// TIA Portal project "babu_3MotorsUsingComparatorsCounters" (V15)

(* hardware
DEVICE "S7-1200 station_1"  S7-1200 Station
   slot 0: "Rack_0"  S7-1200 Rack  Rack  V1.0
   slot 1: "PLC_1"  CPU 1212C DC/DC/DC  6ES7 212-1AE40-0XB0  V4.2
*)

// ===== PLC "PLC_1"  CPU 1212C DC/DC/DC =====

VAR_GLOBAL   // PLC tag table "Default tag table"
   "POWER ON PUSH BUTTON" AT %M0.0 : Bool;
   "POWER ON MEM" AT %M0.1 : Bool;
   "PULSE" AT %M0.2 : Bool;
   "RESTART PULSE" AT %M0.3 : Bool;
   "CYCLE COMPLETE" AT %M0.4 : Bool;
   "RESET COUNTER" AT %M0.5 : Bool;
END_VAR

// folder: System blocks/Program resources

DATA_BLOCK "IEC_Timer_0_DB"   // DB1
{ S7_Optimized_Access := 'TRUE' }
AUTHOR : Simatic
FAMILY : IEC
NAME : IEC_TMR
VERSION : 1.0
// stored: InstanceOfName IEC_TIMER
"IEC_TIMER"
BEGIN
END_DATA_BLOCK

DATA_BLOCK "IEC_Timer_0_DB_1"   // DB2
{ S7_Optimized_Access := 'TRUE' }
AUTHOR : Simatic
FAMILY : IEC
NAME : IEC_TMR
VERSION : 1.0
// stored: InstanceOfName IEC_TIMER
"IEC_TIMER"
BEGIN
END_DATA_BLOCK

DATA_BLOCK "IEC_Counter_0_DB"   // DB3
{ S7_Optimized_Access := 'TRUE' }
AUTHOR : Simatic
FAMILY : IEC
NAME : CNTR
VERSION : 1.0
// stored: InstanceOfName IEC_COUNTER
"IEC_COUNTER"
BEGIN
END_DATA_BLOCK

DATA_BLOCK "IEC_Timer_0_DB_2"   // DB4
{ S7_Optimized_Access := 'TRUE' }
AUTHOR : Simatic
FAMILY : IEC
NAME : IEC_TMR
VERSION : 1.0
// stored: InstanceOfName IEC_TIMER
"IEC_TIMER"
BEGIN
END_DATA_BLOCK

// folder: (top level)

ORGANIZATION_BLOCK "Main"   // OB1, LAD, ProgramCycle
TITLE = "Main Program Sweep (Cycle)"
{ S7_Optimized_Access := 'TRUE' }
VERSION : 0.1
   VAR_INPUT
      Initial_Call : Bool;   // Initial call of this OB
      Remanence : Bool;   // =True, if remanent data are available
   END_VAR
BEGIN

REGION Network 1
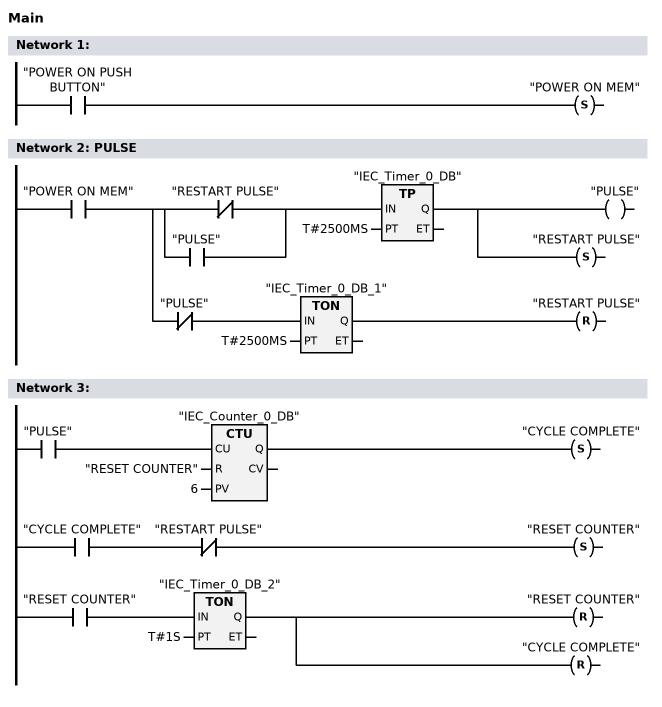
   RUNG wire#powerrail
      Contact( "POWER ON PUSH BUTTON" )
      S_Coil( "POWER ON MEM" )
   END_RUNG
   // the same network as SCL:
   IF "POWER ON PUSH BUTTON" THEN "POWER ON MEM" := TRUE; END_IF;
END_REGION

REGION Network 2: PULSE
   "IEC_Timer_0_DB".TP(IN := "POWER ON MEM" AND (NOT "RESTART PULSE" OR "PULSE"), PT := T#2500MS);
   "PULSE" := "IEC_Timer_0_DB".Q;
   IF "IEC_Timer_0_DB".Q THEN "RESTART PULSE" := TRUE; END_IF;
   "IEC_Timer_0_DB_1".TON(IN := "POWER ON MEM" AND NOT "PULSE", PT := T#2500MS);
   IF "IEC_Timer_0_DB_1".Q THEN "RESTART PULSE" := FALSE; END_IF;
END_REGION

REGION Network 3
   "IEC_Counter_0_DB".CTU(CU := "PULSE", R := "RESET COUNTER", PV := 6);
   IF "IEC_Counter_0_DB".Q THEN "CYCLE COMPLETE" := TRUE; END_IF;
   IF "CYCLE COMPLETE" AND NOT "RESTART PULSE" THEN "RESET COUNTER" := TRUE; END_IF;
   "IEC_Timer_0_DB_2".TON(IN := "RESET COUNTER", PT := T#1S);
   IF "IEC_Timer_0_DB_2".Q THEN
       "RESET COUNTER" := FALSE;
       "CYCLE COMPLETE" := FALSE;
   END_IF;
END_REGION
END_ORGANIZATION_BLOCK